Universal Robots PolyScope program: c_to_g.urp

Program c_to_g (installation=string_planes directory=/programs/string_crossings createdIn=5.17.3 lastSavedIn=5.17.3 robotSerialNumber=20245501435)
Calibrated DH parameters: a=[0.000154, -0.137004, -0.385524, -0.00002, 0.000092, 0]; d=[0.162441, 211.794786, -230.585024, 18.923638, 0.099786, 0.09951]; alpha=[1.569493, -0.001902, 0.003874, 1.570111, -1.570167, 0]; deltaTheta=[0, -1.242934, 1.056292, 0.186646, 0.000002, 0.000001]
InitVariablesNode
Robot Program (runOnlyOnce=true)
  bow_section := -1
  If bow_section≟-1
    MoveJ speed 60 deg/s, acceleration 80 deg/s^2 (useActiveTCP=true) feature=Base
      Waypoint Waypoint_2 (Relative): relativeFromPosition TCP in base x=245.28 y=570.707 z=53.269 mm, rx=-1.8425 ry=-1.3918 rz=0.0687 rad; joints [-132.225, -24.798, 96.315, -169.322, -42.69, -112.608] deg; TCP offset x=28.21 y=-96.107 z=-99.69 mm, rx=0 ry=0 rz=0 rad; TCP in base x=333.315 y=655.493 z=103.665 mm, rx=-1.6491 ry=-1.7982 rz=0.6656 rad; joints [-132.464, -27.758, 71.844, -100.482, -56.043, -147.727] deg
  ElseIf bow_section≟0
    MoveJ speed 60 deg/s, acceleration 80 deg/s^2 (useActiveTCP=true) feature=Base
      Waypoint Waypoint_1 (Relative): relativeFromPosition TCP in base x=195.289 y=411.481 z=21.276 mm, rx=-1.7343 ry=-1.5169 rz=0.4321 rad; joints [-140.232, -30.937, 122.53, -154.989, -45.802, -143.196] deg; TCP in base x=267.77 y=455.818 z=63.349 mm, rx=-1.6064 ry=-1.9107 rz=0.8702 rad; joints [-141.616, -39.193, 108.913, -115.288, -70.781, -159.12] deg
  Else 
    MoveJ speed 60 deg/s, acceleration 80 deg/s^2 (useActiveTCP=true) feature=Base
      Waypoint Waypoint_3 (Relative): relativeFromPosition TCP in base x=152.637 y=275.831 z=-5.997 mm, rx=-1.6121 ry=-1.6008 rz=0.7404 rad; joints [-153.5, -26.651, 138.518, -151.35, -62.643, -165.795] deg; TCP in base x=243.612 y=214.072 z=64.405 mm, rx=-1.5873 ry=-1.9212 rz=0.9621 rad; joints [-169.306, -44.601, 138.125, -133.881, -94.42, -177.775] deg
